PROGRAM AnPart
VAR_INPUT
          iMode                      :INT;
END_VAR

VAR
	fbAnPart: FB_UserMain;
	
END_VAR

CALL();
ACT();

ACTION ACT:
(********模切小时、天产能**********)
(*
aAnDay_date(
EE:=Q104[7],
);
*)
//运行时间统计
Antimedata(
	Month:= PLC_wMonth, 
	dDay:=PLC_wDay , 
	Hour:=PLC_wHour , 
	Mins:=PLC_wMinute , 
	Second:=PLC_wSecond , 
	Alm:=stSysState.bErrorStop AND NOT bAnDoorALM AND 
             NOT (ProductPar.AnPar.MQ.bWindSelect AND  ProductPar.parFilterAD[1].Out_Value<=ProductPar.AnPar.fDiameterAlarm_L) AND 
             NOT( NOT ProductPar.AnPar.MQ.bWindSelect AND  ProductPar.parFilterAD[2].Out_Value<=ProductPar.AnPar.fDiameterAlarm_R), 
	Wait:=(stSysState.iModehmi=2 OR  stSysState.iModehmi=3) AND (NOT stSysState.bErrorStop OR bAnDoorALM ) AND
             NOT (ProductPar.AnPar.MQ.bWindSelect AND  ProductPar.parFilterAD[1].Out_Value<=ProductPar.AnPar.fDiameterAlarm_L) AND 
             NOT( NOT ProductPar.AnPar.MQ.bWindSelect AND  ProductPar.parFilterAD[2].Out_Value<=ProductPar.AnPar.fDiameterAlarm_R) , 
	Run:=stSysState.iModehmi=1  , 
	JP_Wait:=(ProductPar.AnPar.MQ.bWindSelect AND  ProductPar.parFilterAD[1].Out_Value<=ProductPar.AnPar.fDiameterAlarm_L) OR ( NOT ProductPar.AnPar.MQ.bWindSelect AND  ProductPar.parFilterAD[2].Out_Value<=ProductPar.AnPar.fDiameterAlarm_R) , 
	Query:=MQQuery , 
	STTimedata=> , 
	date1:=MQdate );
END_ACTION

ACTION CALL:
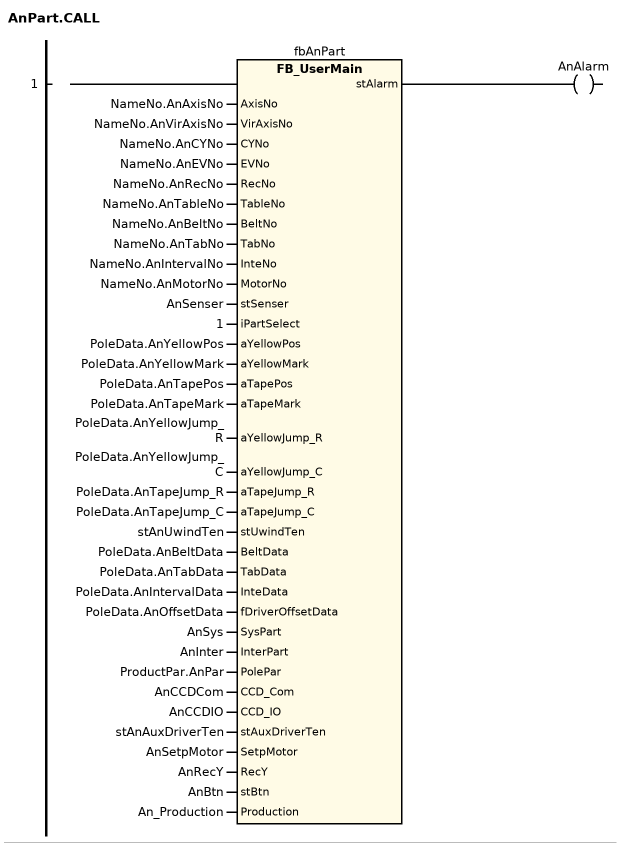
// NETWORK 1
fbAnPart(
    AxisNo := NameNo.AnAxisNo,
    VirAxisNo := NameNo.AnVirAxisNo,
    CYNo := NameNo.AnCYNo,
    EVNo := NameNo.AnEVNo,
    RecNo := NameNo.AnRecNo,
    TableNo := NameNo.AnTableNo,
    BeltNo := NameNo.AnBeltNo,
    TabNo := NameNo.AnTabNo,
    InteNo := NameNo.AnIntervalNo,
    MotorNo := NameNo.AnMotorNo,
    stSenser := AnSenser,
    iPartSelect := 1,
    aYellowPos := PoleData.AnYellowPos,
    aYellowMark := PoleData.AnYellowMark,
    aTapePos := PoleData.AnTapePos,
    aTapeMark := PoleData.AnTapeMark,
    aYellowJump_R := PoleData.AnYellowJump_R,
    aYellowJump_C := PoleData.AnYellowJump_C,
    aTapeJump_R := PoleData.AnTapeJump_R,
    aTapeJump_C := PoleData.AnTapeJump_C,
    stUwindTen := stAnUwindTen,
    BeltData := PoleData.AnBeltData,
    TabData := PoleData.AnTabData,
    InteData := PoleData.AnIntervalData,
    fDriverOffsetData := PoleData.AnOffsetData,
    SysPart := AnSys,
    InterPart := AnInter,
    PolePar := ProductPar.AnPar,
    CCD_Com := AnCCDCom,
    CCD_IO := AnCCDIO,
    stAuxDriverTen := stAnAuxDriverTen,
    SetpMotor := AnSetpMotor,
    RecY := AnRecY,
    stBtn := AnBtn,
    Production := An_Production); // FB_UserMain
AnAlarm := fbAnPart.stAlarm;
END_ACTION

END_PROGRAM

(* stored: Version 1.1.0.1, ProductVersion 3.1.4024.12
   POU AnPart: Id {48a9f71e-029c-4cc9-9718-2b10efec20ea}, SpecialFunc None
   Action ACT: Id {5c1434a3-3d25-4ad4-b518-47976c4c882b}
   Action CALL: Id {e2447a08-8d41-4c98-81c8-648e2c96433c} *)
